{attribute 'hide_all_locals'}
FUNCTION_BLOCK HaltMover IMPLEMENTS ITask
VAR_INPUT
END_VAR
VAR_OUTPUT
END_VAR
VAR
	haltMover : Tc3_McCollisionAvoidance.MC_HaltCA;
	_axis : REFERENCE TO Tc2_MC2.AXIS_REF;
	state : INT;
	_HaltMover : BOOL;
	_busy : BOOL;
	_error : BOOL;
	_done : BOOL;
END_VAR

CASE State OF
	0:
		IF _HaltMover THEN
			_done := FALSE;
			_error := FALSE;
			_busy := TRUE;
			haltMover.Execute := TRUE;
			IF haltMover.Busy THEN
				State := 10;
				_HaltMover := FALSE;
			END_IF
		END_IF
	
	10:
		IF NOT haltMover.Busy THEN
			IF haltMover.Done THEN
				_done := TRUE;
			ELSIF haltMover.Error THEN
				_error := TRUE;
			END_IF
			_busy := FALSE;
			haltMover.Execute := FALSE;
			State := 0;
		END_IF
END_CASE

haltMover(Axis := _axis);

{warning 'add method implementation '}
METHOD Abort : BOOL

VAR
	Position: INT;
END_VAR
haltMover.Execute := FALSE;
_busy := FALSE;
_HaltMover := FALSE;
Abort := TRUE;
State := 0;
END_METHOD

PROPERTY Busy : BOOL
GET
Busy := _busy;
END_GET
END_PROPERTY

PROPERTY Done : BOOL
GET
Done := _done;
END_GET
END_PROPERTY


PROPERTY Error : BOOL
GET
Error := _error;
END_GET
END_PROPERTY

METHOD Execute : BOOL
VAR_INPUT
END_VAR
Execute := _HaltMover := true;
END_METHOD

METHOD FB_init : BOOL
VAR_INPUT
	bInitRetains : BOOL; // if TRUE, the retain variables are initialized (warm start / cold start)
	bInCopyCode : BOOL;  // if TRUE, the instance afterwards gets moved into the copy code (online change)
	axis : reference TO AXIS_REF;
END_VAR
_axis REF= axis;
END_METHOD

END_FUNCTION_BLOCK

(* stored: Version 1.1.0.1, ProductVersion 3.1.4024.6
   POU HaltMover: Id {5e16f656-97ee-4391-96b9-fb1d24ff82ad}, SpecialFunc None
   Method Abort: Id {f69b4fe1-38a5-4078-941d-4d491f1587ae}
   Property Busy: Id {d58d13e4-27b1-4398-a2b2-85f972edbcb8}
   Get Get: Id {926e484f-fb58-45ba-b2e7-ebc79c8e4496}
   Property Done: Id {bcad271f-e2ab-41dc-9338-a4c65d3f42df}
   Get Get: Id {47510195-111c-4e7f-b411-3075dea97802}
   Property Error: Id {b91c58ec-ed1c-4758-91ff-23039261d8ca}
   Get Get: Id {c4421906-7b21-4370-ab3d-09d6277a4ee2}
   Method Execute: Id {671d0ba5-9f92-4fc7-84aa-e5d4dbbeaa24}
   Method FB_init: Id {41479c9c-6cc0-4c29-b41a-fb9449cfb9dd} *)
